// TIA Portal V20 export
TYPE "ASI5_Flags"
   STRUCT
      C1_FlagsFault : Byte;
      C2_FlagsFault : Byte;
   END_STRUCT;
END_TYPE
